(* Schneider Machine Expert - Basic project R15 - Fallback, file version 2.2.0.0 *)
(* ProjectInformations: Name=New project *)

HARDWARE
  Cpu 0: TM221ME16R/G
  EthernetConfiguration: NetworkName=M221, IpAllocationMode=FixedAddress, IpAddress=0.0.0.0, SubnetMask=0.0.0.0
  SerialLineConfiguration: Baud=Baud19200, Parity=ParityEven, DataBits=DataBits8, StopBits=StopBits1, PhysicalMedium=PhysicalMediumRs485, TransmissionMode=TransmissionModeModbusRtu, SlaveId=1, Addressing=SlaveAddressing
  MastTask: UsePeriodScanMode=false, PeriodScan=100
  FastTask: Period=255
  CpuBehavior: StartingMode=StartAsPreviousState, AutoSaveRamOnEeprom=true, WatchdogPeriod=250

SYMBOLS  (address, symbol, comment, settings)
  %S9       SB_FALLBACKOUTPUT  "Set to 1 to apply fallbacks on digital and analog outputs"

POU Process
  (* SectionNumber=1 *)

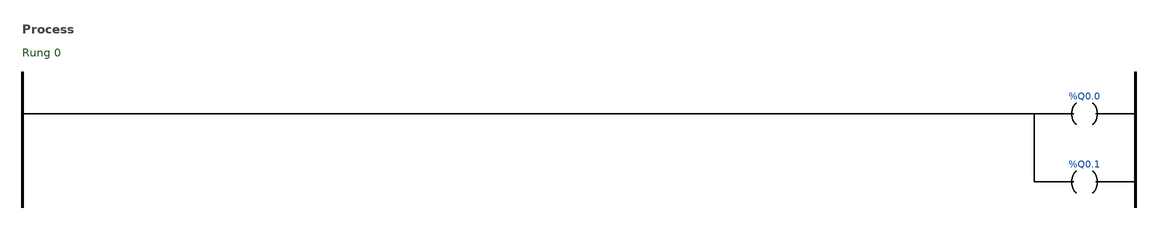

// Rung 0
  LD 1
  ST %Q0.0
  ST %Q0.1
  // as ST:
  //   %Q0.0 := TRUE;
  //   %Q0.1 := TRUE;

POU Config
  (* SectionNumber=2 *)

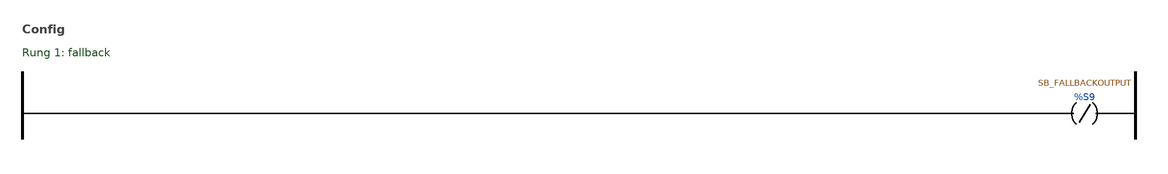

// Rung 1: fallback
  LD 1
  STN %S9                 (* SB_FALLBACKOUTPUT *)
  // as ST:
  //   SB_FALLBACKOUTPUT := FALSE;
